{attribute 'GeneratedUsingTerminal: KL9505-0010'}
{attribute addProperty BoxType "KL9505-0010"}
{attribute addProperty Id "Supply_Voltage_OKAT %I*BOOL0Over_currentAT %I*BOOL0"}
{attribute addProperty CRC "525288819"}
{attribute addProperty Size "0"}
TYPE Diag_1F4F4573 EXTENDS InputBase_8311D824 :
STRUCT
	{attribute addProperty Name "Supply_Voltage_OK"}
	Supply_Voltage_OK AT %I* : BOOL;
	{attribute addProperty Name "Over_current"}
	Over_current AT %I* : BOOL;
END_STRUCT
END_TYPE

(* stored: Version 1.2.0.0, ProductVersion 3.1.4024.9
   DUT Diag_1F4F4573: Id {220fd709-acd2-4ea7-8eb3-043225fe875f} *)
